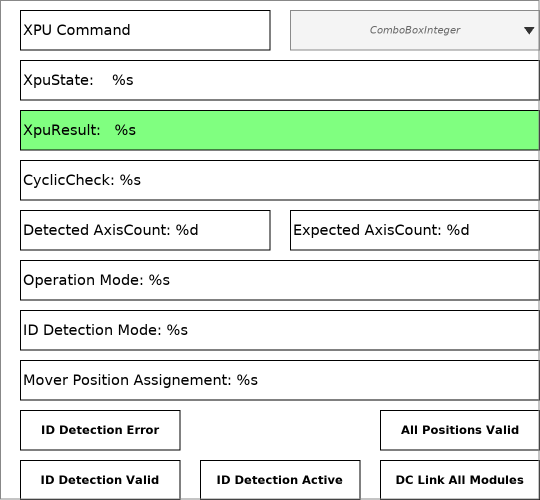
VISUALIZATION XPU_VISU  // 540x500
    Rectangle (20,10 250x40), "XPU Command"
    ComboBoxInteger (290,10 250x40), variable: GVL_XTS.XpuCtrl.Cmd, text list: 'TL_E_CTRL_XPU'
    Rectangle (20,160 520x40), "CyclicCheck: %s", text variable: MAIN.sXpuCheck
    Rectangle (20,60 520x40), "XpuState: %s", text variable: MAIN.sXpuState
    Rectangle (20,110 520x40), "XpuResult: %s", text variable: MAIN.sXpuResult, colour toggle: (MAIN.eXpuResult = E_PROGRESS.PROGRESS_ERROR)
    Rectangle (380,410 160x40), "All Positions Valid", colour toggle: GVL_XTS.XtsTransportState.XpuInfo.AllPositionsValid
    Rectangle (20,410 160x40), "ID Detection Error", colour toggle: GVL_XTS.XtsTransportState.XpuInfo.IdDetectionError
    Rectangle (20,460 160x40), "ID Detection Valid", colour toggle: GVL_XTS.XtsTransportState.XpuInfo.IdDetectionValid
    Rectangle (200,460 160x40), "ID Detection Active", colour toggle: GVL_XTS.XtsTransportState.XpuInfo.IdDetectionActive
    Rectangle (20,260 520x40), "Operation Mode: %s", text variable: MAIN.sXpuOpMode
    Rectangle (20,310 520x40), "ID Detection Mode: %s", text variable: MAIN.sXpuMoverdetectionMode
    Rectangle (20,360 520x40), "Mover Position Assignement: %s", text variable: MAIN.sXpuMoverAssignement
    Rectangle (290,210 250x40), "Expected AxisCount: %d", text variable: GVL_XTS.XtsTransportState.XpuInfo.nExpectedAxisCount
    Rectangle (20,210 250x40), "Detected AxisCount: %d", text variable: GVL_XTS.XtsTransportState.XpuInfo.nDetectedAxisCount
    Rectangle (380,460 160x40), "DC Link All Modules", colour toggle: GVL_XTS.XtsTransportState.XpuState.DcLink
END_VISUALIZATION

(* stored: Version 1.1.0.1, ProductVersion 3.1.4026.12
   Visu XPU_VISU: Id {4496a510-fde6-462f-9a77-f39614139df3} *)
